(* IEC 61131-3 sources: repolevel_ST_code_completion/real_groud_truth最新/repoeval_barrier/readful_result, 13 files *)

(* ---- CAN_Send_Data_SWMC.st ---- *)
VAR
    result : BOOL;
END_VAR

result := FALSE;

// Simulate sending data to the CAN bus
IF (SWMC_ID > 0) AND (id > 0) THEN
    // Here you would typically call a hardware-specific function to send the data
    // For example: CAN_Write(SWMC_ID, id, data);
    result := TRUE; // Assume the data was sent successfully
END_IF;

RETURN result;
END_FUNCTION

// Additional code to handle the CAN communication logic
FUNCTION_BLOCK CAN_Controller
VAR
    sendCounter : UINT;
END_VAR

METHOD Initialize : BOOL
VAR
    success : BOOL;
END_VAR

success := FALSE;

// Initialize the CAN controller
// For example: CAN_Init();

sendCounter := 0;
success := TRUE;

RETURN success;
END_METHOD

METHOD SendData : BOOL
VAR
    success : BOOL;
    sendData : ARRAY[1..8] OF BYTE;
    swmcIdSwitch : UINT;
END_VAR

success := FALSE;

// Example logic for sending data
swmcIdSwitch := sendCounter MOD 2;

CASE swmcIdSwitch OF
    0:
        sendData[1] := WORD_TO_BYTE(gController.sky[3].extendPercent);
        sendData[2] := WORD_TO_BYTE(SHR(gController.sky[3].extendPercent, 8));
        sendData[3] := WORD_TO_BYTE(gController.sky[3].retractPercent);
        sendData[4] := WORD_TO_BYTE(SHR(gController.sky[3].retractPercent, 8));
        sendData[5] := WORD_TO_BYTE(gController.sky[4].extendPercent);
        sendData[6] := WORD_TO_BYTE(SHR(gController.sky[4].extendPercent, 8));
        sendData[7] := WORD_TO_BYTE(gController.sky[4].retractPercent);
        sendData[8] := WORD_TO_BYTE(SHR(gController.sky[4].retractPercent, 8));
        success := CAN_Send_Data_SWMC(1, 16#500, sendData);
    1:
        sendData[1] := WORD_TO_BYTE(gController.sky[5].extendPercent);
        sendData[2] := WORD_TO_BYTE(SHR(gController.sky[5].extendPercent, 8));
        sendData[3] := WORD_TO_BYTE(gController.sky[5].retractPercent);
        sendData[4] := WORD_TO_BYTE(SHR(gController.sky[5].retractPercent, 8));
        sendData[5] := WORD_TO_BYTE(gController.sky[6].extendPercent);
        sendData[6] := WORD_TO_BYTE(SHR(gController.sky[6].extendPercent, 8));
        sendData[7] := WORD_TO_BYTE(gController.sky[6].retractPercent);
        sendData[8] := WORD_TO_BYTE(SHR(gController.sky[6].retractPercent, 8));
        success := CAN_Send_Data_SWMC(1, 16#501, sendData);
END_CASE;

sendCounter := sendCounter + 1;

RETURN success;
END_METHOD

(* ---- CAN_Read_Data_SWMC.st ---- *)
VAR
	receivedFrame : Can_baseframe; // Variable to store the received CAN frame
END_VAR

CASE SWMC_ID OF
	1:
		receivedFrame := gCan.C1RxMsg.RXMsg[I]; // Retrieve data from CAN channel 1
		gCan.C1RxMsg.RxCounter := gCan.C1RxMsg.RxCounter + 1; // Increment the receive counter
	2:
		receivedFrame := gCan.C2RxMsg.RXMsg[I]; // Retrieve data from CAN channel 2
		gCan.C2RxMsg.RxCounter := gCan.C2RxMsg.RxCounter + 1; // Increment the receive counter
	3:
		receivedFrame := gCan.C3RxMsg.RXMsg[I]; // Retrieve data from CAN channel 3
		gCan.C3RxMsg.RxCounter := gCan.C3RxMsg.RxCounter + 1; // Increment the receive counter
	4:
		receivedFrame := gCan.C4RxMsg.RXMsg[I]; // Retrieve data from CAN channel 4
		gCan.C4RxMsg.RxCounter := gCan.C4RxMsg.RxCounter + 1; // Increment the receive counter
	ELSE
		receivedFrame := Can_baseframe(); // Return an empty frame if SWMC_ID is invalid
END_CASE;

RETURN receivedFrame; // Return the received CAN frame

(* ---- CommandExecutor.st ---- *)
VAR
	direct		:TargetDirect;	//方向
END_VAR

CASE direct OF
	TargetDirect.extend:
		CASE level OF
			1:
				gController.grd[idx].extendPercent := REAL_TO_WORD(percent * 65535 / 100);
				gController.grd[idx].retractPercent := 0;
			2:
				gController.sky[idx].extendPercent := REAL_TO_WORD(percent * 65535 / 100);
				gController.sky[idx].retractPercent := 0;
		END_CASE
	TargetDirect.retract:
		CASE level OF
			1:
				gController.grd[idx].extendPercent := 0;
				gController.grd[idx].retractPercent := REAL_TO_WORD(ABS(percent) * 65535 / 100);
			2:
				gController.sky[idx].extendPercent := 0;
				gController.sky[idx].retractPercent := REAL_TO_WORD(ABS(percent) * 65535 / 100);
		END_CASE
	TargetDirect.stop:
		CASE level OF
			1:
				gController.grd[idx].extendPercent := 0;
				gController.grd[idx].retractPercent := 0;
			2:
				gController.sky[idx].extendPercent := 0;
				gController.sky[idx].retractPercent := 0;
		END_CASE
END_CASE

(* ---- CommandExecutor0.st ---- *)
VAR
END_VAR

IF direct = TargetDirect.Extend THEN
	CASE level OF
		1:
			gController.grd[idx].extendPercent := REAL_TO_WORD(percent * 65535 / 100);
			gController.grd[idx].retractPercent := 0;
		2:
			gController.sky[idx].extendPercent := REAL_TO_WORD(percent * 65535 / 100);
			gController.sky[idx].retractPercent := 0;
	END_CASE
ELSIF direct = TargetDirect.Retract THEN
	CASE level OF
		1:
			gController.grd[idx].extendPercent := 0;
			gController.grd[idx].retractPercent := REAL_TO_WORD(percent * 65535 / 100);
		2:
			gController.sky[idx].extendPercent := 0;
			gController.sky[idx].retractPercent := REAL_TO_WORD(percent * 65535 / 100);
	END_CASE
END_IF

(* ---- DataReverse_cmdReverse.st ---- *)
VAR_OUTPUT
	result		:TargetDirect;
END_VAR

IF input = TargetDirect.extend THEN
	result := TargetDirect.retract;
ELSIF input = TargetDirect.retract THEN
	result := TargetDirect.extend;
ELSE
	result := input; // Default case, return the input as is
END_IF;
```

This continuation completes the `cmdReverse` function by adding an output variable `result` and implementing the logic to reverse the `TargetDirect` input. If the input is neither `extend` nor `retract`, it defaults to returning the input unchanged.

(* ---- fileSave_close.st ---- *)
VAR
	lineCount	: INT;
	fileHandle  : DWORD;
	fileName	: STRING;
	datetime	: DATE_AND_TIME;
	UdIntms 	: UDINT;
	UdMsOffset  : UDINT;
	DTimer_Str  : STRING;
	uiYear 		: UINT;
	uiMonth 	: UINT;
	uiDay 		: UINT;
	uiHour 		: UINT;
	uiMinute 	: UINT;
	uiSecond 	: UINT;
	uiMsSecond	: UINT;
END_VAR
VAR_OUTPUT
END_VAR

IF fileHandle = 0 THEN
	datetime := SysTimeGetDateAndTime();
	uiYear := DT_TO_DATE(datetime).year;
	uiMonth := DT_TO_DATE(datetime).month;
	uiDay := DT_TO_DATE(datetime).day;
	uiHour := DT_TO_TIME(datetime).hour;
	uiMinute := DT_TO_TIME(datetime).minute;
	uiSecond := DT_TO_TIME(datetime).second;
	uiMsSecond := DT_TO_TIME(datetime).millisecond;

	DTimer_Str := concat(INT_TO_STRING(uiYear), '_');
	DTimer_Str := concat(DTimer_Str, INT_TO_STRING(uiMonth));
	DTimer_Str := concat(DTimer_Str, '_');
	DTimer_Str := concat(DTimer_Str, INT_TO_STRING(uiDay));
	DTimer_Str := concat(DTimer_Str, '_');
	DTimer_Str := concat(DTimer_Str, INT_TO_STRING(uiHour));
	DTimer_Str := concat(DTimer_Str, '_');
	DTimer_Str := concat(DTimer_Str, INT_TO_STRING(uiMinute));
	DTimer_Str := concat(DTimer_Str, '_');
	DTimer_Str := concat(DTimer_Str, INT_TO_STRING(uiSecond));

	fileName := concat(filePath, '/');
	fileName := concat(fileName, DTimer_Str);
	fileName := concat(fileName, '.txt');

	fileHandle := SysFileOpen(fileName, 'w', F_err);
	IF F_err <> 0 THEN
		fileHandle := 0;
	END_IF;
END_IF;

(* ---- fileSave_createDir.st ---- *)
VAR
	lineCount	: INT;
	fileHandle  : DWORD;
	fileName	: STRING;
	fileHandle0 : DWORD;
	datetime	: DATE_AND_TIME;
	UdIntms 	: UDINT;
	UdMsOffset  : UDINT;
	DTimer_Str  : STRING;
	uiYear 		: UINT;
	uiMonth 	: UINT;
	uiDay 		: UINT;
	uiHour 		: UINT;
	uiMinute 	: UINT;
	uiSecond 	: UINT;
	uiMsSecond	: UINT;

	S_Time64		: SysTime64;
	STT				: CurTimeEx;
	S_Time			: SystemTimeDate;
	Time_Str		: STRING;
	F_err			: DWORD;
	F_HANDL			: DWORD;
END_VAR
VAR_OUTPUT
END_VAR

STT(SystemTime:= S_Time64, TimeDate:= S_Time);

IF fileHandle = 0 THEN
	datetime := SysTimeGetDateAndTime();
	uiYear := datetime.YEAR;
	uiMonth := datetime.MONTH;
	uiDay := datetime.DAY;
	uiHour := datetime.HOUR;
	uiMinute := datetime.MINUTE;
	uiSecond := datetime.SECOND;
	uiMsSecond := datetime.MILLISECOND;

	Time_Str := concat(INT_TO_STRING(uiYear), '-');
	Time_Str := concat(Time_Str, INT_TO_STRING(uiMonth));
	Time_Str := concat(Time_Str, '-');
	Time_Str := concat(Time_Str, INT_TO_STRING(uiDay));
	Time_Str := concat(Time_Str, '_');
	Time_Str := concat(Time_Str, INT_TO_STRING(uiHour));
	Time_Str := concat(Time_Str, '-');
	Time_Str := concat(Time_Str, INT_TO_STRING(uiMinute));
	Time_Str := concat(Time_Str, '-');
	Time_Str := concat(Time_Str, INT_TO_STRING(uiSecond));

	fileName := concat(filePath, '/');
	fileName := concat(fileName, devName);
	fileName := concat(fileName, '_');
	fileName := concat(fileName, Time_Str);
	fileName := concat(fileName, '.txt');

	fileHandle := SysFileOpen(fileName, 'w', F_err);
	IF F_err <> 0 THEN
		fileHandle := 0;
	END_IF;
END_IF;

(* ---- fileSave_new.st ---- *)
VAR
	lineCount	: INT;
	fileHandle  : DWORD;
	fileName	: STRING;
	fileHandle0 : DWORD;
	datetime	: DATE_AND_TIME;
	UdIntms 	: UDINT;
	UdMsOffset  : UDINT;
	DTimer_Str  : STRING;
	uiYear 		: UINT;
	uiMonth 	: UINT;
	uiDay 		: UINT;
	uiHour 		: UINT;
	uiMinute 	: UINT;
	uiSecond 	: UINT;
	uiMsSecond	: UINT;

	S_Time64		: SysTime64;
	STT				: CurTimeEx;
	S_Time			: SystemTimeDate;
	Time_Str		: STRING;
	F_err			: DWORD;
	F_HANDL			: DWORD;
END_VAR
VAR_OUTPUT
END_VAR

STT(SystemTime := S_Time64, TimeDate := S_Time);

IF fileHandle = 0 THEN
	datetime := SysTimeGetDateAndTime();
	uiYear := datetime.YEAR;
	uiMonth := datetime.MONTH;
	uiDay := datetime.DAY;
	uiHour := datetime.HOUR;
	uiMinute := datetime.MINUTE;
	uiSecond := datetime.SECOND;
	uiMsSecond := datetime.MILLISECOND;

	DTimer_Str := concat(INT_TO_STRING(uiYear), '_');
	DTimer_Str := concat(DTimer_Str, INT_TO_STRING(uiMonth));
	DTimer_Str := concat(DTimer_Str, '_');
	DTimer_Str := concat(DTimer_Str, INT_TO_STRING(uiDay));
	DTimer_Str := concat(DTimer_Str, '_');
	DTimer_Str := concat(DTimer_Str, INT_TO_STRING(uiHour));
	DTimer_Str := concat(DTimer_Str, '_');
	DTimer_Str := concat(DTimer_Str, INT_TO_STRING(uiMinute));
	DTimer_Str := concat(DTimer_Str, '_');
	DTimer_Str := concat(DTimer_Str, INT_TO_STRING(uiSecond));
	DTimer_Str := concat(DTimer_Str, '_');
	DTimer_Str := concat(DTimer_Str, INT_TO_STRING(uiMsSecond));

	fileName := concat(filePath, '/');
	fileName := concat(fileName, devName);
	fileName := concat(fileName, '_');
	fileName := concat(fileName, DTimer_Str);
	fileName := concat(fileName, '.txt');

	F_HANDL := SysFileOpen(fileName, 'w', F_err);
	IF F_err = 0 THEN
		fileHandle := F_HANDL;
		lineCount := 0;
	ELSE
		fileHandle := 0;
	END_IF;
END_IF;

(* ---- fileSave_write.st ---- *)
VAR
	lineCount	: INT;
	fileHandle  : DWORD;
	fileName	: STRING;
	data		: STRING;
	F_err		: DWORD;
	tempInt		: INT;
END_VAR
VAR_OUTPUT
END_VAR

# Check if the file handle is valid
IF fileHandle = 0 THEN
	# Attempt to open the file for writing
	fileHandle := SysFileOpen(filePath, 'w', F_err);
	IF F_err <> 0 THEN
		# Handle file open error
		RETURN;
	END_IF;
END_IF;

# Increment the line count and calculate the time interval
lineCount := lineCount + 1;
tempInt := lineCount * intervalt;

# Construct the data string
data := INT_TO_STRING(lineCount);
data := concat(data, '$T$T');
data := concat(data, INT_TO_STRING(tempInt));
IF tempInt < 1000 THEN
	data := concat(data, '$T');
END_IF;
data := concat(data, '$T$T');
data := concat(data, INT_TO_STRING(positionInt));
data := concat(data, '$T');
data := concat(data, INT_TO_STRING(speedInt));
data := concat(data, '$T');
data := concat(data, INT_TO_STRING(stateInt));
data := concat(data, '$R');

# Write the data to the file
SysFileWrite(hFile := fileHandle, pData := ADR(data), size := SIZEOF(data), F_err);
IF F_err <> 0 THEN
	# Handle file write error
	RETURN;
END_IF;

# Optionally close the file if needed
IF lineCount >= 100 THEN
	SysFileClose(hFile := fileHandle);
	fileHandle := 0;
END_IF;

(* ---- mdbsLogicToPhy.st ---- *)
It seems like you are working with a Modbus-related system and defining logic for mapping between physical and logical indices for different sections. Based on the provided code fragments, I will continue writing the `mdbsLogicToPhy` function block to complete the logic for mapping logical indices to physical indices.

```st
VAR
END_VAR

(**
 * 输入华中地址编号，返回本地索引编号
 *)
CASE section OF
    1: // 区域限定(1:skyExtend)
        CASE lgcIdx OF
            10:
                phyIdx := 1;  // sky1e -> 横1
                level := 2;   // 天轨
                direct := TargetDirect.Horizontal;
            11:
                phyIdx := 2;  // sky2e -> 横2
                level := 2;   // 天轨
                direct := TargetDirect.Horizontal;
            12:
                phyIdx := 3;  // sky3e -> 横3
                level := 2;   // 天轨
                direct := TargetDirect.Horizontal;
            13:
                phyIdx := 4;  // sky4e -> 横4
                level := 2;   // 天轨
                direct := TargetDirect.Horizontal;
            14:
                phyIdx := 5;  // sky5e -> 横5
                level := 2;   // 天轨
                direct := TargetDirect.Horizontal;
            15:
                phyIdx := 6;  // sky6e -> 横6
                level := 2;   // 天轨
                direct := TargetDirect.Horizontal;
            16:
                phyIdx := 7;  // sky7e -> 横7
                level := 2;   // 天轨
                direct := TargetDirect.Horizontal;
            17:
                phyIdx := 8;  // sky8e -> 横8
                level := 2;   // 天轨
                direct := TargetDirect.Horizontal;
            18:
                phyIdx := 9;  // sky9e -> 横9
                level := 2;   // 天轨
                direct := TargetDirect.Horizontal;
            19:
                phyIdx := 10; // sky10e -> 横10
                level := 2;   // 天轨
                direct := TargetDirect.Horizontal;
        END_CASE
    2: // 区域限定(2:skyRetract)
        CASE lgcIdx OF
            20:
                phyIdx := 1;  // sky1r -> 纵1
                level := 2;   // 天轨
                direct := TargetDirect.Vertical;
            21:
                phyIdx := 2;  // sky2r -> 纵2
                level := 2;   // 天轨
                direct := TargetDirect.Vertical;
            22:
                phyIdx := 3;  // sky3r -> 纵3
                level := 2;   // 天轨
                direct := TargetDirect.Vertical;
            23:
                phyIdx := 4;  // sky4r -> 纵4
                level := 2;   // 天轨
                direct := TargetDirect.Vertical;
            24:
                phyIdx := 5;  // sky5r -> 纵5
                level := 2;   // 天轨
                direct := TargetDirect.Vertical;
            25:
                phyIdx := 6;  // sky6r -> 纵6
                level := 2;   // 天轨
                direct := TargetDirect.Vertical;
            26:
                phyIdx := 7;  // sky7r -> 纵7
                level := 2;   // 天轨
                direct := TargetDirect.Vertical;
            27:
                phyIdx := 8;  // sky8r -> 纵8
                level := 2;   // 天轨
                direct := TargetDirect.Vertical;
            28:
                phyIdx := 9;  // sky9r -> 纵9
                level := 2;   // 天轨
                direct := TargetDirect.Vertical;
            29:
                phyIdx := 10; // sky10r -> 纵10
                level := 2;   // 天轨
                direct := TargetDirect.Vertical;
        END_CASE
    3: // 区域限定(3:groundExtend)
        CASE lgcIdx OF
            223:
                phyIdx := 1;  // grd1e -> 横1
                level := 1;   // 地轨
                direct := TargetDirect.Horizontal;
            231:
                phyIdx := 2;  // grd2e -> 纵1
                level := 1;   // 地轨

(* ---- mdbsNumToIdx.st ---- *)
VAR
END_VAR

(**
 * 将设备编号解析为对应的层级和索引
 * (level:1->地轨	2->天轨)(idx:内存物理地址对应数组索引)
 *)
CASE devNo OF
	1..10: // 地轨设备编号范围
		level := 1; // 地轨
		idx := devNo; // 索引直接对应设备编号
	11..20: // 天轨设备编号范围
		level := 2; // 天轨
		idx := devNo - 10; // 索引为设备编号减去偏移量
ELSE
	// 默认值处理
	level := 0; // 未定义层级
	idx := -1; // 无效索引
END_CASE;

(* ---- mdbsPhyToLogic.st ---- *)
It seems like you are working with a Modbus-related project, and the provided code fragments are written in Structured Text (ST), commonly used in industrial automation systems. Below is the continuation of the `FUNCTION_BLOCK mdbsPhyToLogic` based on the patterns and logic observed in the provided code fragments:

```st
VAR
END_VAR

(**
 * 将内存物理地址索引解析为华中状态地址
 * (lgcIdx: 华中对应的地址)
 *)
CASE section OF
    1: // 区域限定1: grdExt
        CASE phyIdx OF
            1:  lgcIdx := 127;   // 地轨1 -> 华中地址127
            2:  lgcIdx := 128;   // 地轨2 -> 华中地址128
            3:  lgcIdx := 129;   // 地轨3 -> 华中地址129
            4:  lgcIdx := 130;   // 地轨4 -> 华中地址130
            5:  lgcIdx := 131;   // 地轨5 -> 华中地址131
            6:  lgcIdx := 132;   // 地轨6 -> 华中地址132
            7:  lgcIdx := 133;   // 地轨7 -> 华中地址133
            8:  lgcIdx := 134;   // 地轨8 -> 华中地址134
            9:  lgcIdx := 135;   // 地轨9 -> 华中地址135
            10: lgcIdx := 136;   // 地轨10 -> 华中地址136
        END_CASE;

    2: // 区域限定2: grdRet
        CASE phyIdx OF
            1:  lgcIdx := 175;   // 地轨1 -> 华中地址175
            2:  lgcIdx := 176;   // 地轨2 -> 华中地址176
            3:  lgcIdx := 177;   // 地轨3 -> 华中地址177
            4:  lgcIdx := 178;   // 地轨4 -> 华中地址178
            5:  lgcIdx := 179;   // 地轨5 -> 华中地址179
            6:  lgcIdx := 180;   // 地轨6 -> 华中地址180
            7:  lgcIdx := 181;   // 地轨7 -> 华中地址181
            8:  lgcIdx := 182;   // 地轨8 -> 华中地址182
            9:  lgcIdx := 183;   // 地轨9 -> 华中地址183
            10: lgcIdx := 184;   // 地轨10 -> 华中地址184
        END_CASE;

    3: // 区域限定3: skyExt
        CASE phyIdx OF
            1:  lgcIdx := 223;   // 天轨1 -> 华中地址223
            2:  lgcIdx := 224;   // 天轨2 -> 华中地址224
            3:  lgcIdx := 225;   // 天轨3 -> 华中地址225
            4:  lgcIdx := 226;   // 天轨4 -> 华中地址226
            5:  lgcIdx := 227;   // 天轨5 -> 华中地址227
            6:  lgcIdx := 228;   // 天轨6 -> 华中地址228
            7:  lgcIdx := 229;   // 天轨7 -> 华中地址229
            8:  lgcIdx := 230;   // 天轨8 -> 华中地址230
            9:  lgcIdx := 231;   // 天轨9 -> 华中地址231
            10: lgcIdx := 232;   // 天轨10 -> 华中地址232
        END_CASE;

    4: // 区域限定4: skyRet
        CASE phyIdx OF
            1:  lgcIdx := 271;   // 天轨1 -> 华中地址271
            2:  lgcIdx := 272;   // 天轨2 -> 华中地址272
            3:  lgcIdx := 273;   // 天轨3 -> 华中地址273
            4:  lgcIdx := 274;   // 天轨4 -> 华中地址274
            5:  lgcIdx := 275;   // 天轨5 -> 华中地址275
            6:  lgcIdx := 276;   // 天轨6 -> 华中地址276

(* ---- setButtonByDirect.st ---- *)
VAR
    success : BOOL;
END_VAR

CASE direct OF
    TargetDirect.extend:
        CASE level OF
            1: // 地轨
                gController.grd[idx].extendPercent := 65535; // 100% 伸出
                gController.grd[idx].retractPercent := 0;    // 缩回设为 0%
                success := TRUE;
            2: // 天轨
                gController.sky[idx].extendPercent := 65535; // 100% 伸出
                gController.sky[idx].retractPercent := 0;    // 缩回设为 0%
                success := TRUE;
            ELSE
                success := FALSE; // 无效的 level
        END_CASE
    TargetDirect.retract:
        CASE level OF
            1: // 地轨
                gController.grd[idx].extendPercent := 0;    // 伸出设为 0%
                gController.grd[idx].retractPercent := 65535; // 100% 缩回
                success := TRUE;
            2: // 天轨
                gController.sky[idx].extendPercent := 0;    // 伸出设为 0%
                gController.sky[idx].retractPercent := 65535; // 100% 缩回
                success := TRUE;
            ELSE
                success := FALSE; // 无效的 level
        END_CASE
    ELSE
        success := FALSE; // 无效的 direct
END_CASE

setButtonByDirect := success;
